FUNCTION_BLOCK AxesEnablePointingModelProcess EXTENDS BaseProcess
VAR_INPUT
	///Arguments to be set, before writing do_request TRUE
	{attribute 'OPC.UA.DA' := '1'}
	set: AxesEnablePointingModelProcessArgs;
END_VAR
VAR_OUTPUT
	///Arguments in use by the process, if do_request was accepted
	{attribute 'OPC.UA.DA' := '1'}
	{attribute 'OPC.UA.DA.Access' := '1'}
	get: AxesEnablePointingModelProcessArgs;
END_VAR
VAR_IN_OUT
END_VAR
VAR
END_VAR

IF do_request THEN
    do_request_result := request( name := set.name );
    do_request := FALSE;
END_IF;
SUPER^();

{attribute 'TcRpcEnable' := '1'}
METHOD start
VAR_INPUT
	///Name of the pointing model
	name: STRING;
END_VAR
VAR_OUTPUT
END_VAR
VAR_IN_OUT
END_VAR
VAR
END_VAR
THIS^.get.name := name;
THIS^.statuses.busyStatus( isBusy := TRUE );
THIS^.statuses.healthStatus( isGood := TRUE );
END_METHOD

{attribute 'TcRpcEnable' := '1'}
METHOD request : RequestResults
VAR_INPUT
	///Name of the pointing model
	name: STRING;
END_VAR
VAR_OUTPUT
END_VAR
VAR_IN_OUT
END_VAR
VAR
END_VAR
IF THIS^.statuses.enabledStatus.enabled THEN
    THIS^.start( name := name );
    request := RequestResults.ACCEPTED;
ELSE
    request := RequestResults.REJECTED;
END_IF;
END_METHOD

END_FUNCTION_BLOCK

(* stored: Version 1.1.0.1, ProductVersion 3.1.4019.2
   POU AxesEnablePointingModelProcess: Id {bfb91d2e-4dc2-4cb2-b10b-5ce99b1e5984}, SpecialFunc None
   Method start: Id {160112ed-9980-4c83-88af-60296660a169}
   Method request: Id {7639e654-2a8e-4312-bfd2-7e69a133703c} *)
